RoboDK station: Arctos.rdk

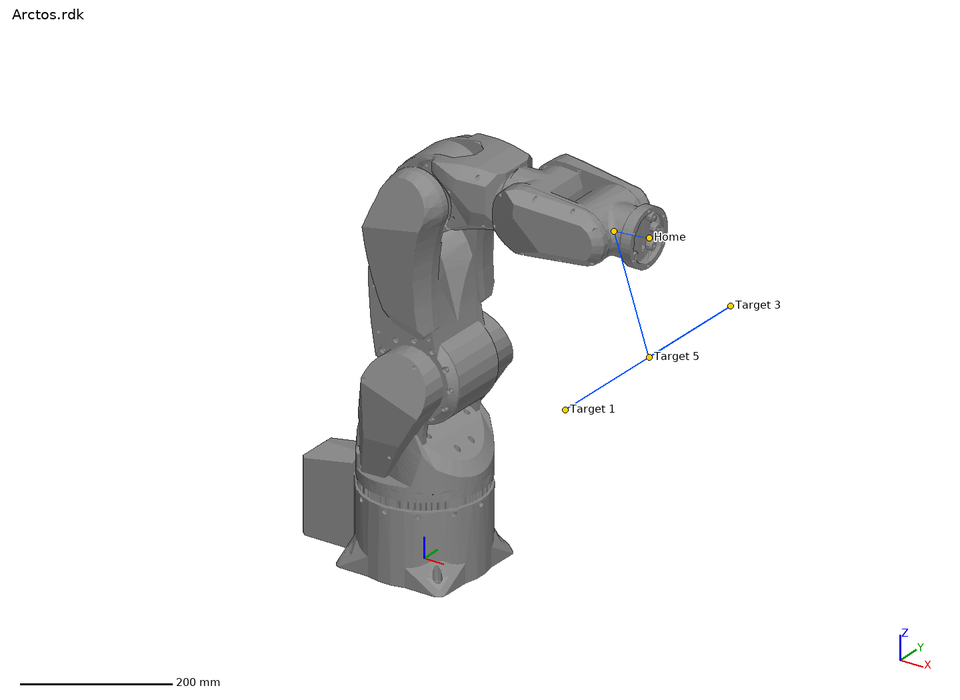
[picture v0: the station drawn from its stored meshes, robots at their saved joint values, targets as dots, program paths as lines]
Station Arctos (saved by RoboDK 5.6.0). Poses are relative to the parent item; angles as X-Y-Z fixed-axis rotations.
  - object b at (0, 0, 0) mm, size 269.1 x 183.6 x 136 mm, geometry from b.step
  - object J1 at (0, 0, 0) mm, size 183.8 x 217.5 x 313.9 mm, geometry from J1.step
  - object J2 (1) at (0, 0, 0) mm, size 144.2 x 196.7 x 374.9 mm, geometry from J2 (1).step
  - object J3 at (0, 0, 0) mm, size 176.8 x 123.2 x 122.2 mm, geometry from J3.step
  - object J4 (1) at (0, 0, 0) mm, size 217.1 x 158.5 x 97.3 mm, geometry from J4 (1).step
  - object J5 at (0, 0, 0) mm, size 118.7 x 78.5 x 80.7 mm, geometry from J5.step
  - object J6 (1) at (0, 0, 0) mm, size 18.5 x 86 x 86 mm, geometry from J6 (1).step
  - frame My Mechanism Base at (899.78, 999.44, 57.25) mm
    - robot Arctos: 6 axes
        modified DH rows (alpha deg, a mm, theta deg, d mm): 0, 0, 0, 287.872; -90, 20.174, -90, 0; 0, 260.986, 0, 0; -90, 19.219, 0, 260.753; 90, 0, 0, 0; -90, 0, 180, 74.745
        joint limits [-200, -125, -50, -200, -100, -200] to [200, 75, 100, 200, 100, 200]; home [0, 0, 0, 0, 0, 0]; saved at [0, -0.971, 0.979, 0.011, 0.008, 0.011]
    - target Home (Cartesian target) at (360.09, 0, 568.08) mm, rotated rx 0 ry 90 rz 0 deg; joints [0, -0.971, 0.979, 0.011, 0.008, 0.011] of Arctos
    - target Target 1 (Cartesian target) at (360.09, -192.34, 394.12) mm, rotated rx 0 ry 90 rz 0 deg; joints [-33.983, -22.516, -12.746, 49.422, -47.385, 38.328] of Arctos
    - target Target 3 (Cartesian target) at (360.09, 186.3, 394.12) mm, rotated rx 0 ry 90 rz 0 deg; joints [33.14, -21.88, -13.662, -48.32, -47.052, -37.425] of Arctos
    - target Target 4 (Cartesian target) at (304.04, 0, 562.49) mm, rotated rx 0 ry 19.94 rz 0 deg; joints [0, -0.684, -16.037, 0, -86.782, 0] of Arctos
    - target Target 5 (Cartesian target) at (360.09, 0, 394.12) mm, rotated rx 0 ry 90 rz 0 deg; joints [0, -11.232, -27.921, 0, -39.154, 0] of Arctos
    - target Target 6 (Cartesian target) at (360.09, 0, 394.12) mm, rotated rx 0 ry 90 rz 0 deg; joints [0, -11.232, -27.921, 0, -39.154, 0] of Arctos
  - program Prog1 (6 instructions, listed below)
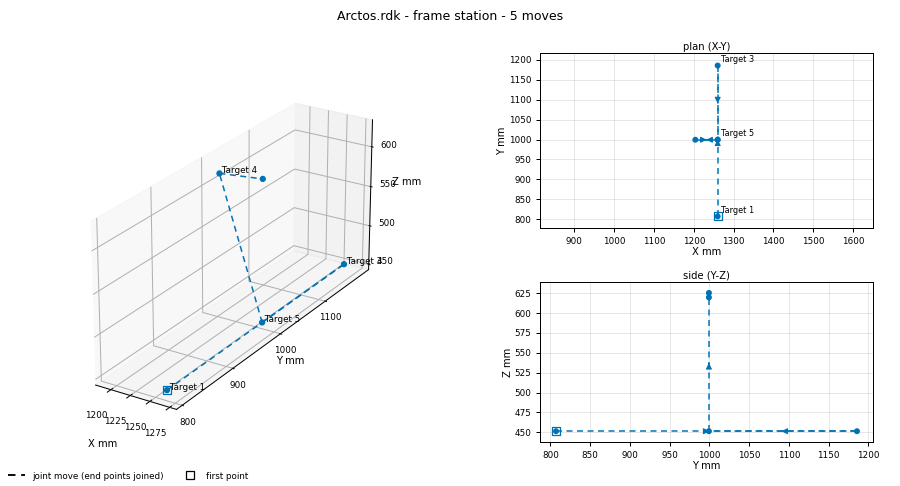
[picture p0: tool path of Arctos.rdk in frame station, 5 of 5 moves have a stored position in this frame; points joined in program order, loops and branches not executed]

--- program Prog1 (robot Arctos) ---
  Set Ref.: My Mechanism Base
  MoveJ (Target 1)
  MoveJ (Target 3)
  MoveJ (Target 5)
  MoveJ (Target 4)
  MoveJ (Home)
